// Core S7.2.1 - the application names its own conditions on this module; the
// library declares none. Safe-motion status (S9.2) is read-only application
// input, so "STO cleared" is declared here by the station that can see it.
// Declared conditions start FALSE: declaring one states an intent to gate.
METHOD DeclareCondition : BOOL
VAR_INPUT
    Index : INT;
    DescriptionKey : STRING(255);
    Reason : E_Reason;
    Bypassable : BOOL;
END_VAR
IF (Index < 1) OR (Index > PL_Fraktal.MAX_PERMINTLK_COND) THEN
    DeclareCondition := FALSE;
    RETURN;
END_IF
_appCond[Index] := FALSE;
DeclareCondition := Intlk.Define(Index := Index, Description := DescriptionKey,
    Reason := Reason, Bypassable := Bypassable);
END_METHOD

// Drive a condition declared by DeclareCondition, every scan.
METHOD SetCondition : BOOL
VAR_INPUT
    Index : INT;
    Ok : BOOL;
END_VAR
IF (Index < 1) OR (Index > PL_Fraktal.MAX_PERMINTLK_COND) THEN
    SetCondition := FALSE;
    RETURN;
END_IF
_appCond[Index] := Ok;
SetCondition := TRUE;
END_METHOD

// §7.6.1 held command - JOG_POS / JOG_NEG. Called EVERY SCAN while the
// operator holds the button; silence stops the axis (see _M_JogCyclic).
//
// This method only RECORDS the request. Nothing moves from here: the decision to
// drive is taken once per scan in _M_JogCyclic, where the interlock, the enabling
// device, the freshness deadline and the command handshake are all weighed
// together. Keeping the decision in one place is what makes it reviewable.
METHOD RequestHeldCommand : BOOL
VAR_INPUT
    Value  : DINT;
    Enable : ST_ManualEnableStatus;
END_VAR
// IF rather than CASE: a CASE label must be a compile-time constant, and
// TO_DINT(enum) is a call. The intent is the same - a defined ELSE (§5.6).
IF Value = TO_DINT(E_AxisCommand.JOG_POS) THEN
    _jogReqDir :=  1;
ELSIF Value = TO_DINT(E_AxisCommand.JOG_NEG) THEN
    _jogReqDir := -1;
ELSE
    // Not a held command of this type. Refuse, and do not record it - an unknown
    // value must never leave a stale direction behind.
    RequestHeldCommand := FALSE;
    RETURN;
END_IF

_jogSeen    := TRUE;
_jogEnabled := Enable.Held;

// Refused up front, with the reason, when no safety-rated enabling device is
// permitting. The axis ALSO has to pass its interlocks in _M_JogCyclic - this is
// an additional requirement, never a way around them (§9).
//
// StationCfg.JogRequiresEnable is what an installation WITHOUT an enabling
// device declares (§3.8a). It relaxes exactly this one requirement: the
// interlocks, the freshness deadline and the command handshake are untouched,
// so a station that declares it still cannot jog through a dropped interlock
// or on a stale request.
IF _station.JogRequiresEnable AND NOT Enable.Held THEN
    OutImm.JogStopReason := PL_ModuleReasons.AXIS_JOG_NOT_ENABLED;
    RequestHeldCommand := FALSE;
    RETURN;
END_IF
RequestHeldCommand := TRUE;
END_METHOD

// The one place a jog is allowed to start, continue, or stop. Runs every scan
// from OnCyclic, whether or not anybody asked - because "nobody asked" is
// precisely the condition that has to stop the axis.
METHOD PRIVATE _M_JogCyclic
VAR
    drive : BOOL;
END_VAR
// Freshness (O10). The timer accumulates while no request arrives, so a caller
// that goes quiet - operator released, HMI closed, network stalled with the
// button still down - stops the axis after JogTimeout. A few scans of jitter are
// tolerated; a dead transport is not.
_tJogStale(IN := NOT _jogSeen, PT := ParCfg.JogTimeout);

// Every gate that must hold for the axis to move by hand, in one expression so
// there is one place to review. Interlocks are NOT bypassed for teaching: the
// station is expected to have wired its guard condition so the safety system's
// teach grant satisfies it, and if it has not, the axis simply does not jog
// (§7.2.1, fail-closed).
drive := (_jogReqDir <> 0)
    AND NOT _tJogStale.Q
    AND (_jogEnabled OR NOT _station.JogRequiresEnable)
    AND Intlk.AllOk
    AND NOT Busy                        // a commanded move owns the axis (§6.1)
    AND __ISVALIDREF(_axis);

// Say why it stopped, once, on the transition. Published status, not an alarm.
IF _jogDriving AND NOT drive THEN
    // The PLC genuinely cannot tell "operator let go" from "link died" - both
    // are simply the request no longer arriving - so it reports what it knows
    // rather than inventing a distinction. The HMI CAN tell, because it knows
    // whether it is still sending, and surfaces the difference there.
    IF _tJogStale.Q THEN
        OutImm.JogStopReason := PL_ModuleReasons.AXIS_JOG_RELEASED;
    ELSIF NOT _jogEnabled AND _station.JogRequiresEnable THEN
        OutImm.JogStopReason := PL_ModuleReasons.AXIS_JOG_NOT_ENABLED;
    ELSIF NOT Intlk.AllOk THEN
        OutImm.JogStopReason := TO_DINT(E_Reason.INTERLOCK_DROPPED);
    ELSE
        OutImm.JogStopReason := PL_ModuleReasons.AXIS_JOG_RELEASED;
    END_IF
    _jogReqDir := 0;
END_IF

IF __ISVALIDREF(_axis) THEN
    _jogFb(Axis := _axis,
           JogForward   := drive AND (_jogReqDir > 0),
           JogBackwards  := drive AND (_jogReqDir < 0),
           Mode         := MC_JOGMODE_CONTINOUS,
           Velocity     := ParCfg.JogVelocity,
           Acceleration := ParCfg.JogAcceleration,
           Deceleration := ParCfg.Deceleration);
END_IF

_jogDriving    := drive;
OutImm.Jogging := drive;
_jogSeen       := FALSE;   // consumed: the caller must ask again next scan
END_METHOD

METHOD Setup : BOOL
VAR_INPUT
    Name    : STRING(80);
    AxisRef : REFERENCE TO AXIS_REF;
    Recipe  : I_RecipeProvider;
END_VAR
VAR
    InitialModel : ST_ModelId;
END_VAR
_M_SetName(Name);
_M_SetPresentation(DisplayNameKey := 'std.moduleType.axis.name', DescriptionKey := 'std.moduleType.axis.description', TypeKey := 'std.moduleType.axis');
_axis REF= AxisRef;                      // [TC3] TC3 S3.11
_recipe := Recipe;
// No Intlk.Define here: safe-motion status and station policy are the
// application's to name (S7.2.1).
_M_PublishCommand(Value := TO_DINT(E_AxisCommand.HOME), Label := 'std.command.home');
_M_PublishCommand(Value := TO_DINT(E_AxisCommand.MOVE_TO), Label := 'std.command.moveTo');
_M_PublishHeldCommand(Value := TO_DINT(E_AxisCommand.JOG_POS), Label := 'std.command.jogPositive');
_M_PublishHeldCommand(Value := TO_DINT(E_AxisCommand.JOG_NEG), Label := 'std.command.jogNegative');
Setup := PrepareRecipe(Model := InitialModel);
IF Setup THEN CommitRecipe(); END_IF

// §3.8b restore, in one call. The rule - version 0 is a first boot that lost
// nothing, any other unrecognized version means a real image was rejected and
// is annunciated with this module's own path - is written ONCE in
// FB_ModuleBase, because every module type with a StationCfg needs exactly it
// (§1.1 O1). This type supplies only the part that is genuinely its own: what
// its declared defaults are.
//
// The CONSEQUENCE of a loss is the deployment's, not this module's: the root
// applies E_ConfigRestorePolicy. Faulting the axis here, as this used to,
// forced BLOCK_UNTIL_ACKNOWLEDGED on every station that ever used an axis.
IF NOT M_RestoreStationCfg(pVersion := ADR(_station.SchemaVersion),
        SchemaVersion := AXIS_STATIONCFG_SCHEMA) THEN
    _station.TaughtPosition := 0.0;          // this type's declared default
    // The default is the SAFE reading: an axis that lost its configuration
    // requires an enabling device again, rather than inheriting a bench's
    // relaxation into a machine that never declared one.
    _station.JogRequiresEnable := TRUE;
END_IF

// §3.8a - the taught position is an ordinary editable value: typeable by an
// engineer who knows the number, and validated against the same soft limits
// whichever way it arrives.
Setup := M_RegisterConfigNumber(Key := 'axis.taughtPosition',
    Item := 'StationCfg/TaughtPosition', LabelKey := 'std.config.axisTaughtPosition',
    Unit := E_EngUnit.MILLIMETER, Kind := E_ConfigKind.STATION_CFG, Storage := E_ConfigStorage.AS_LREAL,
    pTarget := ADR(_station.TaughtPosition), Minimum := ParCfg.SoftMin, Maximum := ParCfg.SoftMax,
    RequiresReady := FALSE) AND Setup;

// §3.8c - and it can be DEMONSTRATED instead of typed: jog the axis to the
// position, then capture. The source is OutImm.ActPos, which this module already
// publishes, so the operator sees the number before storing it (§3.8c(b)).
Setup := M_RegisterCapture(WriteKey := 'axis.taughtPosition',
    pSource := ADR(OutImm.ActPos), SourceStorage := E_ConfigStorage.AS_LREAL) AND Setup;

// §3.8a - published as an editable capability so "does this installation have
// an enabling device?" is visible, audited and carried in a station parameter
// set, instead of being a silent assumption nobody can see.
Setup := M_RegisterConfigFlag(Key := 'axis.jogRequiresEnable',
    Item := 'StationCfg/JogRequiresEnable',
    LabelKey := 'std.config.axisJogRequiresEnable',
    Kind := E_ConfigKind.STATION_CFG, pTarget := ADR(_station.JogRequiresEnable),
    RequiresReady := TRUE) AND Setup;
END_METHOD

// §3.8a/§G.4a - declare whether this INSTALLATION has a safety-rated enabling
// device for manual motion. Called by the composition root; it also stamps the
// schema version forward, so a call made before Setup survives the restore
// (a matching version is restored as-is rather than defaulted).
//
// FALSE relaxes exactly one requirement - the enabling device - and nothing
// else: interlocks, the freshness deadline and the command handshake all still
// apply, and jog still refuses a stale request. A station that declares FALSE
// should declare a §7.5 engineering gate with it, so the machine says out loud
// that it is jogging without one.
METHOD SetJogRequiresEnable : BOOL
VAR_INPUT
    Required : BOOL;
END_VAR
_station.JogRequiresEnable := Required;
_station.SchemaVersion := AXIS_STATIONCFG_SCHEMA;
SetJogRequiresEnable := TRUE;
END_METHOD

// Functional stop used by an owning sequence on abort/interlock loss. This is a
// controlled MC_Stop, NOT a certified safe stop: the safety system remains
// authoritative and STO is its business, not this module's (S9).
METHOD WithdrawOutputs
IF __ISVALIDREF(_axis) THEN
    _moveFb(Axis := _axis, Execute := FALSE);
    _homeFb(Axis := _axis, Execute := FALSE);
    // A held jog is an output of this module like any other, so it is withdrawn
    // here too - otherwise an abort would stop the commanded move and leave a
    // jog running.
    _jogFb(Axis := _axis, JogForward := FALSE, JogBackwards := FALSE);
    _stopFb(Axis := _axis, Execute := TRUE, Deceleration := ParCfg.Deceleration);
END_IF
_jogReqDir  := 0;
_jogDriving := FALSE;
OutImm.Jogging := FALSE;
_tMove(IN := FALSE);
END_METHOD

METHOD PROTECTED OnAbort : DINT
OnAbort := SUPER^.OnAbort();            // base first (S3.14.2)
WithdrawOutputs();
END_METHOD

METHOD PrepareRecipe : BOOL
VAR_INPUT
    Model : ST_ModelId;
END_VAR
IF _recipe = 0 THEN
    _parCfgStaged := ParCfg;
    _recipePrepared := TRUE;
    PrepareRecipe := TRUE;
ELSIF _recipe.Load(ModelCode := Model.ModelCode, RecipeKey := 'AxisCM', pParCfg := ADR(_parCfgStaged), Size := SIZEOF(_parCfgStaged)) THEN
    _recipePrepared := TRUE;
    PrepareRecipe := TRUE;
ELSE
    _M_Fault(E_Reason.RECIPE_INVALID, 'std.error.recipeSchemaInvalid');
    _recipePrepared := FALSE;
    PrepareRecipe := FALSE;
END_IF
END_METHOD

METHOD CommitRecipe
IF _recipePrepared THEN ParCfg := _parCfgStaged; END_IF
_recipePrepared := FALSE;
END_METHOD

METHOD AbortRecipe
_recipePrepared := FALSE;
END_METHOD

// Stop the axis, THEN fault. _M_FaultN raises the reason without touching
// motion, so faulting mid-move would leave the drive commanded - the same defect
// the separator's _M_FaultClosed exists to prevent, and worse here because the
// load is moving.
METHOD PRIVATE _M_FaultStopped
VAR_INPUT
    Code : DINT;
    Text : STRING(255);
END_VAR
WithdrawOutputs();
_M_FaultN(Code := Code, Text := Text);
END_METHOD

METHOD PROTECTED _M_Dispatch
VAR
    dg : ST_Diagnostic;
END_VAR
IF _manualReq THEN
    _manualReq := FALSE;
    IF (_manualCmd = TO_DINT(E_AxisCommand.HOME)) OR (_manualCmd = TO_DINT(E_AxisCommand.MOVE_TO)) THEN
        Command := _manualCmd;
    ELSE
        _M_Fault(E_Reason.UNSUPPORTED_COMMAND, 'std.error.unsupportedAxisCommand');
        RETURN;
    END_IF
END_IF
IF (Command <> E_AxisCommand.HOME) AND (Command <> E_AxisCommand.MOVE_TO) THEN
    _M_Fault(E_Reason.UNSUPPORTED_COMMAND, 'std.error.unsupportedAxisCommand');
    RETURN;
END_IF
IF Command = E_AxisCommand.HOME THEN
    _M_TagCommand(Id := 1, Label := 'std.command.home');          // S8.11.4(a)
ELSE
    _M_TagCommand(Id := 2, Label := 'std.command.moveTo');
END_IF
_M_ApplyConditions();
Intlk();
IF NOT Intlk.AllOk THEN
    // HELD, not a fault (S6.1). Losing a declared condition mid-move is expected
    // - an operator releasing an enable is the designed way to stop. The axis is
    // brought to a controlled stop by the same permit that gates the enable, and
    // the move resumes from step 10 with a full MoveTimeout window so a hold
    // cannot silently consume travel time the axis was not moving for.
    WithdrawOutputs();
    dg := Intlk.Diagnostic;
    dg.SourcePath := _name;                          // owner sets the path (S7.2)
    _M_HoldDiag(Diag := dg);
    _step := 10;
    RETURN;
END_IF
IF Command = E_AxisCommand.HOME THEN
    _M_Home();
ELSE
    _M_MoveTo();
END_IF
END_METHOD

METHOD PRIVATE _M_Home
IF NOT __ISVALIDREF(_axis) THEN
    _M_FaultN(Code := PL_ModuleReasons.AXIS_DRIVE_FAULT, Text := 'std.error.axisNotBound');
    RETURN;
END_IF
CASE _step OF
    10:
        OutCmd.InPosition := FALSE;
        _homed := FALSE;                       // homing invalidates any previous datum
        _homeFb(Axis := _axis, Execute := FALSE);
        _tMove(IN := FALSE);
        _step := 20;
    20:
        _homeFb(Axis := _axis, Execute := TRUE, Position := 0.0, HomingMode := MC_DefaultHoming);
        _tMove(IN := TRUE, PT := ParCfg.HomeTimeout);
        IF _homeFb.Done THEN
            _homeFb(Axis := _axis, Execute := FALSE);
            _tMove(IN := FALSE);
            _homed := TRUE;
            _M_Complete();
        ELSIF _homeFb.Error THEN
            _M_FaultStopped(Code := PL_ModuleReasons.AXIS_DRIVE_FAULT, Text := 'std.error.axisDriveFault');
        ELSIF _homeFb.CommandAborted THEN
            // CommandAborted means another motion command took the axis, which is
            // an abort and not a defect - route it through the base's own abort
            // path rather than inventing a fault for it.
            AbortCommand();
        ELSIF _tMove.Q THEN
            _M_FaultStopped(Code := PL_ModuleReasons.AXIS_MOVE_TIMEOUT, Text := 'std.error.axisMoveTimeout');
        END_IF
ELSE
    _M_Fault(E_Reason.STEP_STALLED, 'std.error.undefinedStep');    // defined ELSE (S5.6)
END_CASE
END_METHOD

METHOD PRIVATE _M_MoveTo
// Validate the REQUEST before the STATE, and both before commanding motion
// (S5.6). Annex G checked homed-first; range-first is used here because a target
// outside the soft limits is malformed regardless of whether the axis is homed,
// and reporting "not homed" for an impossible target sends the operator to the
// wrong problem. It also makes both rejections provable without a licensed NC
// axis, since neither issues an MC_* call.
IF (ParCmd.Target < ParCfg.SoftMin) OR (ParCmd.Target > ParCfg.SoftMax) THEN
    _M_FaultN(Code := PL_ModuleReasons.AXIS_TARGET_OOR, Text := 'std.error.axisTargetOutOfRange');
    RETURN;
END_IF
IF NOT _homed THEN
    _M_FaultN(Code := PL_ModuleReasons.AXIS_NOT_HOMED, Text := 'std.error.axisNotHomed');
    RETURN;
END_IF
IF NOT __ISVALIDREF(_axis) THEN
    _M_FaultN(Code := PL_ModuleReasons.AXIS_DRIVE_FAULT, Text := 'std.error.axisNotBound');
    RETURN;
END_IF
CASE _step OF
    10:
        OutCmd.InPosition := FALSE;
        _moveFb(Axis := _axis, Execute := FALSE);
        _tMove(IN := FALSE);
        _step := 20;
    20:
        // MC_MoveAbsolute's Busy/Done/Error/CommandAborted map one-to-one onto
        // the CM handshake, which is what lets a parent Unit command MOVE_TO
        // exactly as it commands a cylinder EXTEND (S6.1).
        _moveFb(Axis := _axis, Execute := TRUE, Position := ParCmd.Target,
            Velocity := ParCfg.Velocity, Acceleration := ParCfg.Acceleration,
            Deceleration := ParCfg.Deceleration);
        _tMove(IN := TRUE, PT := ParCfg.MoveTimeout);
        IF _moveFb.Done THEN
            _moveFb(Axis := _axis, Execute := FALSE);
            _tMove(IN := FALSE);
            OutCmd.InPosition := TRUE;
            _M_Complete();
        ELSIF _moveFb.Error THEN
            _M_FaultStopped(Code := PL_ModuleReasons.AXIS_DRIVE_FAULT, Text := 'std.error.axisDriveFault');
        ELSIF _moveFb.CommandAborted THEN
            // CommandAborted means another motion command took the axis, which is
            // an abort and not a defect - route it through the base's own abort
            // path rather than inventing a fault for it.
            AbortCommand();
        ELSIF _tMove.Q THEN
            _M_FaultStopped(Code := PL_ModuleReasons.AXIS_MOVE_TIMEOUT, Text := 'std.error.axisMoveTimeout');
        END_IF
ELSE
    _M_Fault(E_Reason.STEP_STALLED, 'std.error.undefinedStep');
END_CASE
END_METHOD

END_FUNCTION_BLOCK

// ---- FB_SeparatorCM.TcPOU
// Annex A worked example on the base class: the type is ONLY its device logic.
//
// It defines NO interlocks of its own, deliberately. Core S7.2.1 confines a
// reusable library to "device-intrinsic conditions or explicitly injected generic
// policy", and none of Annex A's four published conditions qualify: area-safe is
// a S9.2 safety alias, air pressure is a utility, jam is a flag that is not even
// on this device's HAL, and downstream-ready is line policy. All four belong to
// the owning Unit's Release/Permissives object (S7.2.1, S4.2).
//
// So the application declares and drives them through DeclareCondition/
// SetCondition. They land in this module's own FB_PermIntlk, which keeps the
// provenance S7.2.1 requires - first-out, release report and HMI drill-down all
// read the same ST_IntlkCond records - without the library naming policy it
// cannot see. A per-condition setter was rejected: FB_CylinderCM.SetAreaSafe is
// exactly that shape and no application has ever called it.
FUNCTION_BLOCK FB_SeparatorCM EXTENDS FB_ControlModuleBase
VAR_INPUT
    Command : E_SeparatorCommand;
    ParCfg : ST_SeparatorParCfg;
    ParCmd : ST_SeparatorParCmd;
END_VAR
VAR_OUTPUT
    OutCmd : ST_SeparatorOutCmd;
    OutImm : ST_SeparatorOutImm;
    Intlk  : FB_PermIntlk;
END_VAR
VAR
    {attribute 'OPC.UA.DA' := '0'}
    _hal    : REFERENCE TO ST_SeparatorHal;
    {attribute 'OPC.UA.DA' := '0'}
    _recipe : I_RecipeProvider;
    _tPhase : TON;                       // per-phase timeout (open / clear / arrive)
    _tClose : TON;                       // close delay
    _parCfgStaged : ST_SeparatorParCfg;
    _recipePrepared : BOOL;
    // Application-owned conditions (S7.2.1). Declared FALSE so a declared-but-
    // undriven condition holds the module rather than silently permitting it.
    _appCond : ARRAY[1..PL_Fraktal.MAX_PERMINTLK_COND] OF BOOL;
END_VAR

Cyclic();

METHOD PROTECTED OnCyclic : DINT
OnCyclic := SUPER^.OnCyclic();
// Re-drive every application condition each scan, so a manual command obeys the
// same rule as a sequenced one (S7.2).
_M_ApplyConditions();
Intlk();
IF __ISVALIDREF(_hal) THEN              // defensive (S5.6) [TC3]
    OutImm.CarrierAt    := _hal.CarrierAt;
    OutImm.CarrierAfter := _hal.CarrierAfter;
    OutImm.OpenedFb     := _hal.OpenedFb;
    OutImm.ValveOpen    := _hal.ValveOpen;
    OutCmd.SeparatorOpen := _hal.ValveOpen;
END_IF
END_METHOD

METHOD PRIVATE _M_ApplyConditions
VAR
    i : INT;
END_VAR
FOR i := 1 TO PL_Fraktal.MAX_PERMINTLK_COND DO
    Intlk.Cond[i] := _appCond[i];
END_FOR
END_METHOD

// Core S7.2.1 - the application names its own conditions on this module.
// The library defines none, so every index is the application's to claim.
// Returns FALSE on an out-of-range index rather than silently ignoring it (S5.6).
//
// Declared conditions start FALSE: declaring one states an intent to gate, so
// the fail-closed default is to hold until the application drives it. A station
// that wants no gate simply declares nothing.
METHOD DeclareCondition : BOOL
VAR_INPUT
    Index : INT;
    DescriptionKey : STRING(255);
    Reason : E_Reason;
    Bypassable : BOOL;
END_VAR
IF (Index < 1) OR (Index > PL_Fraktal.MAX_PERMINTLK_COND) THEN
    DeclareCondition := FALSE;
    RETURN;
END_IF
_appCond[Index] := FALSE;
DeclareCondition := Intlk.Define(Index := Index, Description := DescriptionKey,
    Reason := Reason, Bypassable := Bypassable);
END_METHOD

// Drive a condition declared by DeclareCondition. Call it every scan from the
// owning Unit's Release object; the value is re-applied in OnCyclic so dispatch
// and the release report always read the same state.
METHOD SetCondition : BOOL
VAR_INPUT
    Index : INT;
    Ok : BOOL;
END_VAR
IF (Index < 1) OR (Index > PL_Fraktal.MAX_PERMINTLK_COND) THEN
    SetCondition := FALSE;
    RETURN;
END_IF
_appCond[Index] := Ok;
SetCondition := TRUE;
END_METHOD

METHOD Setup : BOOL
VAR_INPUT
    Name   : STRING(80);
    HalRef : REFERENCE TO ST_SeparatorHal;
    Recipe : I_RecipeProvider;
END_VAR
VAR
    InitialModel : ST_ModelId;
END_VAR
_M_SetName(Name);
_M_SetPresentation(DisplayNameKey := 'std.moduleType.separator.name', DescriptionKey := 'std.moduleType.separator.description', TypeKey := 'std.moduleType.separator');
_hal REF= HalRef;                        // [TC3] TC3 S3.11
_recipe := Recipe;
// No Intlk.Define here: this type publishes no condition it cannot itself
// derive (S7.2.1). The application declares its own via DeclareCondition.
_M_PublishCommand(Value := TO_DINT(E_SeparatorCommand.SEPARATE), Label := 'std.command.separate');
_M_PublishCommand(Value := TO_DINT(E_SeparatorCommand.OPEN_CLOSE), Label := 'std.command.openClose');
Setup := PrepareRecipe(Model := InitialModel);
IF Setup THEN CommitRecipe(); END_IF
END_METHOD

// Functional stop used by an owning sequence on abort/interlock loss.
// This is not a certified stop; the safety system remains authoritative (S9).
METHOD WithdrawOutputs
IF __ISVALIDREF(_hal) THEN
    _hal.ValveOpen := FALSE;
END_IF
END_METHOD

METHOD PROTECTED OnAbort : DINT
OnAbort := SUPER^.OnAbort();            // base first (S3.14.2)
IF __ISVALIDREF(_hal) THEN
    _hal.ValveOpen := FALSE;
END_IF
END_METHOD

METHOD PrepareRecipe : BOOL
VAR_INPUT
    Model : ST_ModelId;
END_VAR
IF _recipe = 0 THEN
    _parCfgStaged := ParCfg;
    _recipePrepared := TRUE;
    PrepareRecipe := TRUE;
ELSIF _recipe.Load(ModelCode := Model.ModelCode, RecipeKey := 'SeparatorCM', pParCfg := ADR(_parCfgStaged), Size := SIZEOF(_parCfgStaged)) THEN
    _recipePrepared := TRUE;
    PrepareRecipe := TRUE;
ELSE
    _M_Fault(E_Reason.RECIPE_INVALID, 'std.error.recipeSchemaInvalid');
    _recipePrepared := FALSE;
    PrepareRecipe := FALSE;
END_IF
END_METHOD

METHOD CommitRecipe
IF _recipePrepared THEN ParCfg := _parCfgStaged; END_IF
_recipePrepared := FALSE;
END_METHOD

METHOD AbortRecipe
_recipePrepared := FALSE;
END_METHOD

METHOD PROTECTED _M_Dispatch
VAR
    dg : ST_Diagnostic;
END_VAR
IF _manualReq THEN
    _manualReq := FALSE;
    IF (_manualCmd = TO_DINT(E_SeparatorCommand.SEPARATE)) OR (_manualCmd = TO_DINT(E_SeparatorCommand.OPEN_CLOSE)) THEN
        Command := _manualCmd;
    ELSE
        _M_Fault(E_Reason.UNSUPPORTED_COMMAND, 'std.error.unsupportedSeparatorCommand');
        RETURN;
    END_IF
END_IF
IF (Command <> E_SeparatorCommand.SEPARATE) AND (Command <> E_SeparatorCommand.OPEN_CLOSE) THEN
    _M_Fault(E_Reason.UNSUPPORTED_COMMAND, 'std.error.unsupportedSeparatorCommand');
    RETURN;
END_IF
IF Command = E_SeparatorCommand.SEPARATE THEN
    _M_TagCommand(Id := 1, Label := 'std.command.separate');      // S8.11.4(a)
ELSE
    _M_TagCommand(Id := 2, Label := 'std.command.openClose');
END_IF
_M_ApplyConditions();
Intlk();
IF NOT Intlk.AllOk THEN
    // HELD, not a fault (S6.1): an interlock is a condition that must hold DURING
    // the action, and losing one is often expected - the same reasoning as
    // FB_CylinderCM. Outputs are withdrawn here by the same permit that gates
    // them; only the classification and the way out differ. Rewinding to step 10
    // re-arms the phase timer with a full window, so a hold cannot silently
    // consume travel time the carrier was not moving for.
    IF __ISVALIDREF(_hal) THEN
        _hal.ValveOpen := FALSE;
    END_IF
    _tPhase(IN := FALSE);
    dg := Intlk.Diagnostic;
    dg.SourcePath := _name;                          // owner sets the path (S7.2)
    _M_HoldDiag(Diag := dg);
    _step := 10;
    RETURN;
END_IF
IF Command = E_SeparatorCommand.OPEN_CLOSE THEN
    _M_OpenClose();
    RETURN;
END_IF
// ---- SEPARATE: release exactly one carrier (Annex A) ----------------------
CASE _step OF
    10:                                  // open, and require a carrier present
        OutCmd.SeparateOk := FALSE;
        _hal.ValveOpen := TRUE;
        _tPhase(IN := TRUE, PT := ParCfg.MaxOpenTime);
        IF _hal.CarrierAt THEN
            _tPhase(IN := FALSE);
            _step := 20;
        ELSIF _tPhase.Q THEN
            _tPhase(IN := FALSE);
            _M_FaultClosed(Code := PL_ModuleReasons.SEP_NO_CARRIER_AT, Text := 'std.error.separatorNoCarrierAt');
        END_IF
    20:                                  // the carrier must clear CarrierAt
        _tPhase(IN := TRUE, PT := ParCfg.MaxOpenTime);
        IF NOT _hal.CarrierAt THEN
            _tPhase(IN := FALSE);
            IF ParCfg.CheckAfter THEN _step := 30; ELSE _step := 40; END_IF
        ELSIF _tPhase.Q THEN
            _tPhase(IN := FALSE);
            _M_FaultClosed(Code := PL_ModuleReasons.SEP_CARRIER_NOT_CLEARED, Text := 'std.error.separatorCarrierNotCleared');
        END_IF
    30:                                  // arrival check past the separator
        _tPhase(IN := TRUE, PT := ParCfg.SOnMaxTime);
        IF _hal.CarrierAfter THEN
            _tPhase(IN := FALSE);
            _step := 40;
        ELSIF _tPhase.Q THEN
            _tPhase(IN := FALSE);
            _M_FaultClosed(Code := PL_ModuleReasons.SEP_CARRIER_NOT_ARRIVED, Text := 'std.error.separatorCarrierNotArrived');
        END_IF
    40:                                  // close after the configured delay
        _tClose(IN := TRUE, PT := ParCfg.CloseDelay);
        IF _tClose.Q OR (ParCfg.CloseDelay = T#0S) THEN
            _tClose(IN := FALSE);
            _hal.ValveOpen := FALSE;
            IF ParCfg.CheckAfter THEN
                _tPhase(IN := TRUE, PT := ParCfg.SOnMaxTime);
                _step := 50;
            ELSE
                OutCmd.SeparateOk := TRUE;
                _M_Complete();
            END_IF
        END_IF
    50:                                  // the carrier must clear CarrierAfter
        _tPhase(IN := TRUE, PT := ParCfg.SOnMaxTime);
        IF NOT _hal.CarrierAfter THEN
            _tPhase(IN := FALSE);
            OutCmd.SeparateOk := TRUE;
            _M_Complete();
        ELSIF _tPhase.Q THEN
            _tPhase(IN := FALSE);
            _M_FaultClosed(Code := PL_ModuleReasons.SEP_SON_NOT_CLEARED, Text := 'std.error.separatorSonNotCleared');
        END_IF
ELSE
    _M_Fault(E_Reason.STEP_STALLED, 'std.error.undefinedStep');    // defined ELSE (S5.6)
END_CASE
END_METHOD

METHOD PRIVATE _M_OpenClose
// Hold the stopper open or closed. Closing is immediate; opening optionally
// confirms the feedback when the station has wired one (ParCfg.UsesOpenFb).
_hal.ValveOpen := ParCmd.OpenStopper;
IF NOT ParCmd.OpenStopper THEN
    _tPhase(IN := FALSE);
    _M_Complete();
    RETURN;
END_IF
IF NOT ParCfg.UsesOpenFb THEN
    _tPhase(IN := FALSE);
    _M_Complete();
    RETURN;
END_IF
_tPhase(IN := TRUE, PT := ParCfg.MaxOpenTime);
IF _hal.OpenedFb THEN
    _tPhase(IN := FALSE);
    _M_Complete();
ELSIF _tPhase.Q THEN
    _tPhase(IN := FALSE);
    _M_FaultClosed(Code := PL_ModuleReasons.SEP_NOT_OPENED_FB, Text := 'std.error.separatorNotOpenedFb');
END_IF
END_METHOD

// Withdraw the valve, THEN fault. _M_FaultN only raises the reason; it does not
// touch outputs, so faulting from an open phase would leave the stopper
// energised while the module reported ERROR. Annex A faults and closes in one
// step for exactly this reason, and a separator that stays open on a fault
// keeps releasing carriers it can no longer account for.
METHOD PRIVATE _M_FaultClosed
VAR_INPUT
    Code : DINT;
    Text : STRING(255);
END_VAR
WithdrawOutputs();
_M_FaultN(Code := Code, Text := Text);
END_METHOD

END_FUNCTION_BLOCK

// ---- FB_ConfigurableCylinderCM.TcPOU
// Production-grade basic pneumatic cylinder Control Module (Core §2.2 base) with
// OPTIONAL and REDUNDANT position sensors (safety cylinders). Per position: 0..N
// sensors; 0 = sensorless (time-based). 'Arrived' = ALL present sensors TRUE (AND,
// safest); a persistent split of redundant sensors faults (discrepancy monitoring).
// The type is ONLY its device logic; lifecycle/timing/first-out/abort are inherited.
FUNCTION_BLOCK FB_ConfigurableCylinderCM EXTENDS FB_ControlModuleBase
VAR_INPUT
    Command : E_ConfigurableCylinderCommand;
    ParCfg : ST_ConfigurableCylinderParCfg;
    ParCmd : ST_ConfigurableCylinderParCmd;
END_VAR
VAR_OUTPUT
    OutCmd : ST_ConfigurableCylinderOutCmd;
    OutImm : ST_ConfigurableCylinderOutImm;
    Intlk  : FB_PermIntlk;
END_VAR
VAR
    {attribute 'OPC.UA.DA' := '0'}
    _hal     : REFERENCE TO ST_ConfigurableCylinderHal;
    {attribute 'OPC.UA.DA' := '0'}
    _recipe  : I_RecipeProvider;
    _tMove   : TON;
    _tSettle : TON;
    _tDiscH  : TON;                             // home discrepancy timer
    _tDiscW  : TON;                             // work discrepancy timer
    _cfgOk   : BOOL;
    _areaSafe : BOOL := TRUE;                   // §7.2 application-supplied area/process interlock
    _areaSafeKey : STRING(255);
    _parCfgStaged : ST_ConfigurableCylinderParCfg;
    _recipePrepared : BOOL;
END_VAR

Cyclic();

METHOD Setup : BOOL
VAR_INPUT
    Name   : STRING(80);
    HalRef : REFERENCE TO ST_ConfigurableCylinderHal;
    Recipe : I_RecipeProvider;
END_VAR
VAR
    InitialModel : ST_ModelId;
END_VAR
_M_SetName(Name);
_M_SetPresentation(DisplayNameKey := 'std.moduleType.configurableCylinder.name', DescriptionKey := 'std.moduleType.configurableCylinder.description', TypeKey := 'std.moduleType.configurableCylinder');
_M_PublishCommand(Value := TO_DINT(E_ConfigurableCylinderCommand.TO_HOME), Label := 'std.command.toHome');   // §7.6.1 catalog
_M_PublishCommand(Value := TO_DINT(E_ConfigurableCylinderCommand.TO_WORK), Label := 'std.command.toWork');
_hal REF= HalRef;                                        // [TC3] TC3 §3.11
_recipe := Recipe;
Intlk.Define(Index := 1, Description := 'std.interlock.areaSafe', Reason := E_Reason.INTERLOCK_DROPPED, Bypassable := FALSE);
Setup := PrepareRecipe(Model := InitialModel);
IF Setup THEN CommitRecipe(); END_IF
END_METHOD

METHOD PrepareRecipe : BOOL
VAR_INPUT
    Model : ST_ModelId;
END_VAR
_parCfgStaged := ParCfg;
IF _recipe <> 0 THEN
    IF NOT _recipe.Load(ModelCode := Model.ModelCode, RecipeKey := 'ConfigurableCylinderCM', pParCfg := ADR(_parCfgStaged), Size := SIZEOF(_parCfgStaged)) THEN
        _M_Fault(E_Reason.RECIPE_INVALID, 'std.error.recipeSchemaInvalid');
        PrepareRecipe := FALSE;
        RETURN;
    END_IF
END_IF
// counts within [0..MAX]; sensorless direction needs a usable travel time
_cfgOk := (_parCfgStaged.HomeSensorCount >= 0) AND (_parCfgStaged.HomeSensorCount <= PL_Fraktal.MAX_POS_SENSORS)
      AND (_parCfgStaged.WorkSensorCount >= 0) AND (_parCfgStaged.WorkSensorCount <= PL_Fraktal.MAX_POS_SENSORS)
      AND (_parCfgStaged.TravelTime < _parCfgStaged.MoveTimeout)
      AND ((_parCfgStaged.HomeSensorCount > 0) OR (_parCfgStaged.TravelTime > T#0S))
      AND ((_parCfgStaged.WorkSensorCount > 0) OR (_parCfgStaged.TravelTime > T#0S));
IF NOT _cfgOk THEN
    _M_FaultN(PL_ModuleReasons.CYL_CFG_INVALID, 'std.error.cylinderConfigurationInvalid');
    PrepareRecipe := FALSE;
    RETURN;
END_IF
_recipePrepared := TRUE;
PrepareRecipe := TRUE;
END_METHOD

METHOD CommitRecipe
IF _recipePrepared THEN ParCfg := _parCfgStaged; END_IF
_recipePrepared := FALSE;
END_METHOD

METHOD AbortRecipe
_recipePrepared := FALSE;
END_METHOD

// TRUE iff EVERY wired sensor for the position reads TRUE (AND-combine, safest).
// Count = 0 -> not sensor-decided (caller uses the time path).
METHOD PROTECTED _M_PosArrived : BOOL
VAR_INPUT
    Work : BOOL;    // TRUE = work position, FALSE = home
END_VAR
VAR
    i, n : INT;
    all  : BOOL;
END_VAR
n := SEL(Work, ParCfg.HomeSensorCount, ParCfg.WorkSensorCount);
IF n <= 0 THEN
    _M_PosArrived := FALSE;      // no sensors: caller must use the time-based path
    RETURN;
END_IF
all := TRUE;
FOR i := 1 TO n DO
    IF Work THEN
        IF NOT _hal.WorkFb[i] THEN all := FALSE; END_IF
    ELSE
        IF NOT _hal.HomeFb[i] THEN all := FALSE; END_IF
    END_IF
END_FOR
_M_PosArrived := all;
END_METHOD

// TRUE iff the position's redundant sensors DISAGREE (at least one TRUE and at
// least one FALSE) — the discrepancy condition. Single/zero sensor => never split.
METHOD PROTECTED _M_PosSplit : BOOL
VAR_INPUT
    Work : BOOL;
END_VAR
VAR
    i, n : INT;
    anyT, anyF : BOOL;
END_VAR
n := SEL(Work, ParCfg.HomeSensorCount, ParCfg.WorkSensorCount);
IF n < 2 THEN
    _M_PosSplit := FALSE;
    RETURN;
END_IF
FOR i := 1 TO n DO
    IF Work THEN
        IF _hal.WorkFb[i] THEN anyT := TRUE; ELSE anyF := TRUE; END_IF
    ELSE
        IF _hal.HomeFb[i] THEN anyT := TRUE; ELSE anyF := TRUE; END_IF
    END_IF
END_FOR
_M_PosSplit := anyT AND anyF;
END_METHOD

// live position resolve + discrepancy monitoring (both positions, every scan)
METHOD PROTECTED OnCyclic : DINT
OnCyclic := SUPER^.OnCyclic();
Intlk.Cond[1] := _areaSafe;
Intlk();
IF NOT __ISVALIDREF(_hal) THEN
    RETURN;
END_IF
OutImm.AtHome := (ParCfg.HomeSensorCount > 0) AND _M_PosArrived(Work := FALSE);
OutImm.AtWork := (ParCfg.WorkSensorCount > 0) AND _M_PosArrived(Work := TRUE);

// discrepancy monitoring — a persistent split of redundant sensors is a fault
_tDiscH(IN := _M_PosSplit(Work := FALSE), PT := ParCfg.DiscrepancyTime);
_tDiscW(IN := _M_PosSplit(Work := TRUE),  PT := ParCfg.DiscrepancyTime);
IF (_tDiscH.Q OR _tDiscW.Q) AND (_exec <> E_ExecState.ERROR) THEN
    _M_FaultN(PL_ModuleReasons.CYL_DISCREPANCY, 'std.error.cylinderSensorDiscrepancy');
END_IF

// resolve position (AtHome/AtWork already AND-combined)
IF OutImm.AtHome AND OutImm.AtWork THEN
    OutImm.Position := E_CylinderPosition.UNKNOWN;
ELSIF OutImm.AtHome THEN OutImm.Position := E_CylinderPosition.HOME;
ELSIF OutImm.AtWork THEN OutImm.Position := E_CylinderPosition.WORK;
ELSIF (ParCfg.HomeSensorCount > 0) OR (ParCfg.WorkSensorCount > 0) THEN OutImm.Position := E_CylinderPosition.MID;
END_IF

// both-positions-active plausibility while idle
IF (_exec = E_ExecState.READY) AND OutImm.AtHome AND OutImm.AtWork THEN
    _M_FaultN(PL_ModuleReasons.CYL_POS_IMPLAUSIBLE, 'std.error.cylinderPositionImplausible');
END_IF
END_METHOD

// §3.14.2 — fail-safe abort
METHOD PROTECTED OnAbort : DINT
OnAbort := SUPER^.OnAbort();
IF NOT __ISVALIDREF(_hal) THEN
    RETURN;
END_IF
IF ParCfg.DeenergizeOnAbort THEN
    _hal.ToWorkOut := FALSE;
    _hal.ToHomeOut := FALSE;
ELSIF ParCfg.SafePosOnAbort = E_CylinderPosition.WORK THEN
    _hal.ToWorkOut := TRUE;  _hal.ToHomeOut := FALSE;
ELSE
    _hal.ToWorkOut := FALSE; _hal.ToHomeOut := NOT ParCfg.SingleActing;
END_IF
END_METHOD

// Core §7.2/§7.2.1 — the application supplies this type's area/process interlock,
// the same shape as SetDirectionalPermits: a method (not an OPC UA write), and the
// condition is re-evaluated every scan so a manual command obeys the same rule.
//
// This replaces a SIM-only force hook that used to drive Cond[1] directly. That
// hook was the ONLY writer of the condition, so the slot an operator sees as
// "area safe" could be moved by a test and by nothing else: a reusable type
// published an interlock its application had no way to supply (§7.2.1), and the
// bypass shipped in every release build (§5.7). Driving the real condition is
// also strictly better test evidence - T3 now exercises the shipped path.
//
// Defaults TRUE: a station that declares no area interlock is not gated by one.
METHOD SetAreaSafe
VAR_INPUT
    Ok : BOOL;
    DescriptionKey : STRING(255);
END_VAR
_areaSafe := Ok;
_areaSafeKey := DescriptionKey;
IF _areaSafeKey <> '' THEN
    Intlk.Define(Index := 1, Description := _areaSafeKey, Reason := E_Reason.INTERLOCK_DROPPED, Bypassable := FALSE);
ELSE
    ;
END_IF
END_METHOD

// drive -> await (all-sensors-agree, or time when sensorless) -> settle -> done
METHOD PROTECTED _M_Dispatch
VAR
    toWork  : BOOL;
    n       : INT;
    arrived : BOOL;
    d       : ST_Diagnostic;
END_VAR
IF _manualReq THEN
    _manualReq := FALSE;                        // §7.6.1: apply the manual command value
    Command := _manualCmd;                      // routed THROUGH dispatch — interlocks still apply
END_IF
IF (Command <> E_ConfigurableCylinderCommand.TO_HOME) AND (Command <> E_ConfigurableCylinderCommand.TO_WORK) THEN
    _M_Fault(E_Reason.UNSUPPORTED_COMMAND, 'std.error.unsupportedCylinderCommand');
    RETURN;
END_IF
IF Command = E_ConfigurableCylinderCommand.TO_WORK THEN
    _M_TagCommand(Id := 2, Label := 'std.command.toWork');
    toWork := TRUE;
ELSE
    _M_TagCommand(Id := 1, Label := 'std.command.toHome');
    toWork := FALSE;
END_IF
IF NOT Intlk.AllOk THEN
    _hal.ToWorkOut := FALSE;
    _hal.ToHomeOut := FALSE;
    d := Intlk.Diagnostic;
    d.SourcePath := _name;
    _M_FaultDiag(d);
    RETURN;
END_IF
n := SEL(toWork, ParCfg.HomeSensorCount, ParCfg.WorkSensorCount);   // sensors on the TARGET position
CASE _step OF
    10:
        OutCmd.ReachedPosition := E_CylinderPosition.UNKNOWN;
        _hal.ToWorkOut := toWork;
        _hal.ToHomeOut := (NOT toWork) AND (NOT ParCfg.SingleActing);
        _tMove(IN := FALSE);
        _tSettle(IN := FALSE);
        _step := 20;
    20:  // await arrival
        _tMove(IN := TRUE, PT := ParCfg.MoveTimeout);
        IF n > 0 THEN
            arrived := _M_PosArrived(Work := toWork);        // ALL sensors agree
        ELSE
            _tSettle(IN := TRUE, PT := ParCfg.TravelTime);      // sensorless -> travel time
            arrived := _tSettle.Q;
        END_IF
        IF arrived THEN
            _tSettle(IN := FALSE);
            _step := 30;
        ELSIF _tMove.Q THEN
            _tMove(IN := FALSE);
            _M_FaultN(SEL(toWork, PL_ModuleReasons.CYL_HOME_NOT_REACHED, PL_ModuleReasons.CYL_WORK_NOT_REACHED),
                      SEL(toWork, 'std.error.cylinderHomeTimeout', 'std.error.cylinderWorkTimeout'));
        END_IF
    30:  // settle/debounce; re-confirm all sensors still agree
        _tSettle(IN := TRUE, PT := ParCfg.SettleTime);
        IF n <= 0 THEN
            OutCmd.ReachedPosition := SEL(toWork, E_CylinderPosition.HOME, E_CylinderPosition.WORK);
            _M_Complete();
        ELSIF _M_PosArrived(Work := toWork) THEN
            IF _tSettle.Q THEN
                OutCmd.ReachedPosition := SEL(toWork, E_CylinderPosition.HOME, E_CylinderPosition.WORK);
                _M_Complete();
            END_IF
        ELSE
            _tSettle(IN := FALSE);
            _step := 20;                                     // lost agreement; keep waiting in MoveTimeout
        END_IF
ELSE
    _M_Fault(E_Reason.STEP_STALLED, 'std.error.undefinedStep');
END_CASE
END_METHOD

PROPERTY AtPos : E_CylinderPosition
GET
AtPos := OutImm.Position;
END_GET
END_PROPERTY

END_FUNCTION_BLOCK

// ---- FB_ConfigurableCylinderSim.TcPOU
// §5.7 sim plant for FB_ConfigurableCylinderCM with redundant sensors: after a travel time
// it sets all HomeFb[1..HomeN] / WorkFb[1..WorkN] together. StuckWork[i]/StuckHome[i]
// pin a sensor OFF so a test can inject a discrepancy.
FUNCTION_BLOCK FB_ConfigurableCylinderSim
VAR_INPUT
    Travel : TIME := T#100MS;
    HomeN  : INT := 1;
    WorkN  : INT := 1;
    StuckHome : ARRAY[1..PL_Fraktal.MAX_POS_SENSORS] OF BOOL;   // TRUE = pin this sensor OFF
    StuckWork : ARRAY[1..PL_Fraktal.MAX_POS_SENSORS] OF BOOL;
END_VAR
VAR
    {attribute 'OPC.UA.DA' := '0'}
    _hal : REFERENCE TO ST_ConfigurableCylinderHal;
    _tW, _tH : TON;
    i : INT;
END_VAR

IF NOT __ISVALIDREF(_hal) THEN
    RETURN;
END_IF
_tW(IN := _hal.ToWorkOut, PT := Travel);
IF _tW.Q THEN
    FOR i := 1 TO WorkN DO _hal.WorkFb[i] := NOT StuckWork[i]; END_FOR
    FOR i := 1 TO HomeN DO _hal.HomeFb[i] := FALSE; END_FOR
END_IF
_tH(IN := _hal.ToHomeOut OR (NOT _hal.ToWorkOut AND NOT _hal.ToHomeOut), PT := Travel);
IF _tH.Q THEN
    FOR i := 1 TO HomeN DO _hal.HomeFb[i] := NOT StuckHome[i]; END_FOR
    FOR i := 1 TO WorkN DO _hal.WorkFb[i] := FALSE; END_FOR
END_IF

METHOD Setup : BOOL
VAR_INPUT
    HalRef : REFERENCE TO ST_ConfigurableCylinderHal;
    TravelTime : TIME;
    Home : INT;
    Work : INT;
END_VAR
VAR
    j : INT;
END_VAR
_hal REF= HalRef;
Travel := TravelTime;
HomeN := Home;
WorkN := Work;
FOR j := 1 TO HomeN DO _hal.HomeFb[j] := TRUE; END_FOR   // start at home, all agree
Setup := TRUE;
END_METHOD

END_FUNCTION_BLOCK

// ---- FB_ClampEM.TcPOU
// Annex B on the EM base: orchestration only, no device logic (§3.5); rollup §8.2.
FUNCTION_BLOCK FB_ClampEM EXTENDS FB_EquipmentModuleBase
VAR_INPUT
    Command : E_ClampCommand;
    ParCfg : ST_ClampParCfg;
    ParCmd : ST_ClampParCmd;
END_VAR
VAR_OUTPUT
    CylA, CylB : FB_CylinderCM;
    OutCmd : ST_ClampOutCmd;
    OutImm : ST_ClampOutImm;
END_VAR
VAR
    {attribute 'OPC.UA.DA' := '0'}
    _recipe : I_RecipeProvider;
    _tSettle : TON;
    _parCfgStaged : ST_ClampParCfg;
    _recipePrepared : BOOL;
END_VAR

Cyclic();

METHOD PROTECTED OnCyclic : DINT
OnCyclic := SUPER^.OnCyclic();
_M_TickChildren();                       // children stay live (Annex B §B.3)
END_METHOD

METHOD PrepareRecipe : BOOL
VAR_INPUT
    Model : ST_ModelId;
END_VAR
IF _recipe = 0 THEN
    _parCfgStaged := ParCfg;
    _recipePrepared := TRUE;
ELSIF _recipe.Load(ModelCode := Model.ModelCode, RecipeKey := 'ClampEM', pParCfg := ADR(_parCfgStaged), Size := SIZEOF(_parCfgStaged)) THEN
    _recipePrepared := TRUE;
ELSE
    _M_Fault(E_Reason.RECIPE_INVALID, 'std.error.recipeSchemaInvalid');
    _recipePrepared := FALSE;
    PrepareRecipe := FALSE;
    RETURN;
END_IF
PrepareRecipe := SUPER^.PrepareRecipe(Model := Model);
IF NOT PrepareRecipe THEN _recipePrepared := FALSE; END_IF
END_METHOD

METHOD CommitRecipe
SUPER^.CommitRecipe();
IF _recipePrepared THEN ParCfg := _parCfgStaged; END_IF
_recipePrepared := FALSE;
END_METHOD

METHOD AbortRecipe
SUPER^.AbortRecipe();
_recipePrepared := FALSE;
END_METHOD

METHOD Setup : BOOL
VAR_INPUT
    Name : STRING(80);
    HalA : REFERENCE TO ST_CylinderHal;
    HalB : REFERENCE TO ST_CylinderHal;
    Recipe : I_RecipeProvider;
END_VAR
VAR
    InitialModel : ST_ModelId;
END_VAR
_M_SetName(Name);
_M_SetPresentation(DisplayNameKey := 'std.moduleType.clamp.name', DescriptionKey := 'std.moduleType.clamp.description', TypeKey := 'std.moduleType.clamp');
_recipe := Recipe;
CylA.Setup(Name := CONCAT(Name, '.CylA'), HalRef := HalA, Recipe := Recipe);
CylB.Setup(Name := CONCAT(Name, '.CylB'), HalRef := HalB, Recipe := Recipe);
_M_Register(CylA);
_M_Register(CylB);
_M_PublishCommand(Value := TO_DINT(E_ClampCommand.CLAMP), Label := 'std.command.clamp');
_M_PublishCommand(Value := TO_DINT(E_ClampCommand.UNCLAMP), Label := 'std.command.unclamp');
Setup := PrepareRecipe(Model := InitialModel);
IF Setup THEN CommitRecipe(); END_IF
END_METHOD

METHOD PROTECTED _M_Dispatch
VAR
    dir : E_CylinderCommand;
    ext : BOOL;
END_VAR
IF _manualReq THEN
    _manualReq := FALSE;
    IF (_manualCmd = TO_DINT(E_ClampCommand.CLAMP)) OR (_manualCmd = TO_DINT(E_ClampCommand.UNCLAMP)) THEN
        Command := _manualCmd;
    ELSE
        _M_Fault(E_Reason.UNSUPPORTED_COMMAND, 'std.error.unsupportedClampCommand');
        RETURN;
    END_IF
END_IF
IF (Command <> E_ClampCommand.CLAMP) AND (Command <> E_ClampCommand.UNCLAMP) THEN
    _M_Fault(E_Reason.UNSUPPORTED_COMMAND, 'std.error.unsupportedClampCommand');
    RETURN;
END_IF
ext := (Command = E_ClampCommand.CLAMP);
dir := SEL(ext, E_CylinderCommand.RETRACT, E_CylinderCommand.EXTEND);
IF ext THEN
    _M_TagCommand(Id := 1, Label := 'std.command.clamp');
ELSE
    _M_TagCommand(Id := 2, Label := 'std.command.unclamp');
END_IF
CASE _step OF
    10:  // command both cylinders in parallel (Annex B)
        OutCmd.Confirmed := FALSE;
        CylA.Abort := FALSE;
        CylB.Abort := FALSE;
        CylA.Command := dir;
        CylB.Command := dir;
        CylA.Execute := TRUE;
        CylB.Execute := TRUE;
        _tSettle(IN := FALSE);
        _step := 20;
    20:  // join on both Done — roll up the first child Error, or its HELD reason (§8.2)
        IF CylA.Error OR CylB.Error THEN
            _M_RollupFault();
            CylA.Abort := TRUE;                    // stop the partner safely
            CylB.Abort := TRUE;
            CylA.Execute := FALSE;
            CylB.Execute := FALSE;
        ELSIF CylA.Held OR CylB.Held THEN
            // §6.1 HELD — a child is waiting on a named condition, not broken. Keep
            // the join open and adopt its reason so the EM is held-and-explained
            // instead of silently BUSY; both children resume by themselves. The
            // partner keeps its command: aborting it would turn a recoverable wait
            // into the half-finished clamp this join exists to prevent.
            _M_RollupHold();
        ELSIF CylA.Done AND CylB.Done THEN
            CylA.Execute := FALSE;
            CylB.Execute := FALSE;
            _step := 30;
        END_IF
    30:  // settle, then confirm both feedbacks held (EM-level check, Annex B)
        _tSettle(IN := TRUE, PT := ParCfg.SettleTime);
        IF _tSettle.Q THEN
            _tSettle(IN := FALSE);
            IF (ext AND CylA.OutImm.Extended AND CylB.OutImm.Extended)
            OR ((NOT ext) AND CylA.OutImm.Retracted AND CylB.OutImm.Retracted) THEN
                OutImm.Clamped   := ext;
                OutImm.Unclamped := NOT ext;
                OutCmd.Confirmed := TRUE;
                _M_Complete();
            ELSE
                _M_FaultN(PL_ModuleReasons.CLAMP_NOT_CONFIRMED, 'std.error.clampNotConfirmedAfterSettle');
            END_IF
        END_IF
ELSE
    _M_Fault(E_Reason.STEP_STALLED, 'std.error.undefinedStep');
END_CASE
END_METHOD

END_FUNCTION_BLOCK

// ---- FB_CylinderCM.TcPOU
// Annex A/B pattern on the base class: the type is ONLY its device logic.
FUNCTION_BLOCK FB_CylinderCM EXTENDS FB_ControlModuleBase
VAR_INPUT
    Command : E_CylinderCommand;
    ParCfg : ST_CylinderParCfg;
    ParCmd : ST_CylinderParCmd;
END_VAR
VAR_OUTPUT
    OutCmd : ST_CylinderOutCmd;
    OutImm : ST_CylinderOutImm;
    Intlk  : FB_PermIntlk;
END_VAR
VAR
    {attribute 'OPC.UA.DA' := '0'}
    _hal    : REFERENCE TO ST_CylinderHal;
    {attribute 'OPC.UA.DA' := '0'}
    _recipe : I_RecipeProvider;
    _tMove  : TON;
    _areaSafe : BOOL := TRUE;           // §7.2 application-supplied area/process interlock
    _areaSafeKey : STRING(255);
    _parCfgStaged : ST_CylinderParCfg;
    _recipePrepared : BOOL;
    _directionPermitsConfigured : BOOL;
    _extendPermit, _retractPermit : BOOL := TRUE;
    _extendPermitKey, _retractPermitKey : STRING(255);
    _extendedSensorTag, _retractedSensorTag : STRING(80);
    _extendedSensorAddress, _retractedSensorAddress : STRING(80);
    _extendOutputTag, _retractOutputTag : STRING(80);
    _extendedTimeoutKey, _retractedTimeoutKey, _bothSensorsKey : STRING(255);
    _bothSensorTags, _bothSensorAddresses : STRING(80);
END_VAR

Cyclic();

METHOD PROTECTED OnCyclic : DINT
OnCyclic := SUPER^.OnCyclic();
Intlk.Cond[1] := _areaSafe;             // §7.2 area-safe/air-ok, supplied via SetAreaSafe
IF NOT _directionPermitsConfigured OR (Command = E_CylinderCommand.NONE) THEN
    Intlk.Cond[2] := TRUE;
ELSIF Command = E_CylinderCommand.EXTEND THEN
    Intlk.Cond[2] := _extendPermit;
ELSIF Command = E_CylinderCommand.RETRACT THEN
    Intlk.Cond[2] := _retractPermit;
ELSE
    Intlk.Cond[2] := FALSE;
END_IF
Intlk();
IF __ISVALIDREF(_hal) THEN              // defensive (§5.6) [TC3]
    OutImm.Extended  := _hal.ExtendedFb;
    OutImm.Retracted := _hal.RetractedFb;
END_IF
OutImm.ExtendedSensorTag := _extendedSensorTag;
OutImm.RetractedSensorTag := _retractedSensorTag;
OutImm.ExtendOutputTag := _extendOutputTag;
OutImm.RetractOutputTag := _retractOutputTag;
END_METHOD

// Schematic identity is application configuration, not device behavior.
// Diagnostics keep SourcePath as this module and add the exact failed channel.
METHOD ConfigureIoIdentity
VAR_INPUT
    Identity : ST_CylinderIoIdentity;
END_VAR
_extendedSensorTag := Identity.ExtendedSensor.Tag;
_extendedSensorAddress := Identity.ExtendedSensor.Address;
_retractedSensorTag := Identity.RetractedSensor.Tag;
_retractedSensorAddress := Identity.RetractedSensor.Address;
_extendOutputTag := Identity.ExtendOutput.Tag;
_retractOutputTag := Identity.RetractOutput.Tag;
_extendedTimeoutKey := Identity.ExtendedTimeoutKey;
_retractedTimeoutKey := Identity.RetractedTimeoutKey;
_bothSensorsKey := Identity.BothSensorsKey;
_bothSensorTags := CONCAT(Identity.ExtendedSensor.Tag, CONCAT(' / ', Identity.RetractedSensor.Tag));
_bothSensorAddresses := CONCAT(Identity.ExtendedSensor.Address, CONCAT(' / ', Identity.RetractedSensor.Address));
END_METHOD

// Functional stop used by an owning sequence on abort/interlock loss.
// This is not a certified stop; the safety system remains authoritative.
METHOD WithdrawOutputs
IF __ISVALIDREF(_hal) THEN
    _hal.ExtendOut := FALSE;
    _hal.RetractOut := FALSE;
END_IF
END_METHOD

// Symmetric counterpart to WithdrawOutputs, for an owning sequence that withdrew a
// cylinder to hold a phase and now wants it driving again — a press dwell whose
// two-hand button was released and re-pressed, where the force comes from the valve
// latched by the already-completed EXTEND, so nothing else would re-energize it.
// Re-asserts ONLY the last commanded direction and ONLY while that direction's own
// permit is satisfied, so it can never restore an output the interlock is withholding:
// the caller asks, this module still decides. Idempotent; safe to call every scan.
// Not a certified enable — the safety system remains authoritative (§9).
METHOD RestoreOutputs
VAR
    permitted : BOOL;
END_VAR
IF NOT __ISVALIDREF(_hal) THEN
    RETURN;
END_IF
IF Command = E_CylinderCommand.EXTEND THEN
    permitted := _extendPermit OR NOT _directionPermitsConfigured;
ELSIF Command = E_CylinderCommand.RETRACT THEN
    permitted := _retractPermit OR NOT _directionPermitsConfigured;
ELSE
    permitted := FALSE;                 // no direction commanded: nothing to restore (§5.6)
END_IF
IF NOT permitted OR NOT Intlk.AllOk THEN
    RETURN;
END_IF
_hal.ExtendOut  := (Command = E_CylinderCommand.EXTEND);
_hal.RetractOut := (Command = E_CylinderCommand.RETRACT);
END_METHOD

METHOD PROTECTED OnAbort : DINT
OnAbort := SUPER^.OnAbort();            // base first (§3.14.2)
IF __ISVALIDREF(_hal) THEN
    _hal.ExtendOut := FALSE;
    _hal.RetractOut := FALSE;
END_IF
END_METHOD

METHOD PrepareRecipe : BOOL
VAR_INPUT
    Model : ST_ModelId;
END_VAR
IF _recipe = 0 THEN
    _parCfgStaged := ParCfg;
    _recipePrepared := TRUE;
    PrepareRecipe := TRUE;
ELSIF _recipe.Load(ModelCode := Model.ModelCode, RecipeKey := 'CylinderCM', pParCfg := ADR(_parCfgStaged), Size := SIZEOF(_parCfgStaged)) THEN
    _recipePrepared := TRUE;
    PrepareRecipe := TRUE;
ELSE
    _M_Fault(E_Reason.RECIPE_INVALID, 'std.error.recipeSchemaInvalid');
    _recipePrepared := FALSE;
    PrepareRecipe := FALSE;
END_IF
END_METHOD

METHOD CommitRecipe
IF _recipePrepared THEN ParCfg := _parCfgStaged; END_IF
_recipePrepared := FALSE;
END_METHOD

METHOD AbortRecipe
_recipePrepared := FALSE;
END_METHOD

METHOD Setup : BOOL
VAR_INPUT
    Name   : STRING(80);
    HalRef : REFERENCE TO ST_CylinderHal;
    Recipe : I_RecipeProvider;
END_VAR
VAR
    InitialModel : ST_ModelId;
END_VAR
_M_SetName(Name);
_M_SetPresentation(DisplayNameKey := 'std.moduleType.cylinder.name', DescriptionKey := 'std.moduleType.cylinder.description', TypeKey := 'std.moduleType.cylinder');
_hal REF= HalRef;                        // [TC3] TC3 §3.11
_recipe := Recipe;
// A library type owns a std.* key; an application overrides the text through
// SetAreaSafe when its own condition is more specific (§7.2.1).
Intlk.Define(Index := 1, Description := 'std.interlock.areaSafe', Reason := E_Reason.INTERLOCK_DROPPED, Bypassable := FALSE);
Intlk.Define(Index := 2, Description := 'std.interlock.directionPermitted', Reason := E_Reason.INTERLOCK_DROPPED, Bypassable := FALSE);
_M_PublishCommand(Value := TO_DINT(E_CylinderCommand.EXTEND), Label := 'std.command.extend');
_M_PublishCommand(Value := TO_DINT(E_CylinderCommand.RETRACT), Label := 'std.command.retract');
Setup := PrepareRecipe(Model := InitialModel);
IF Setup THEN CommitRecipe(); END_IF
END_METHOD

// Core §7.2/§7.2.1 — the application supplies this type's area/process interlock,
// the same shape as SetDirectionalPermits: a method (not an OPC UA write), and the
// condition is re-evaluated every scan so a manual command obeys the same rule.
//
// This replaces a SIM-only force hook that used to drive Cond[1] directly. That
// hook was the ONLY writer of the condition, so the slot an operator sees as
// "area safe" could be moved by a test and by nothing else: a reusable type
// published an interlock its application had no way to supply (§7.2.1), and the
// bypass shipped in every release build (§5.7). Driving the real condition is
// also strictly better test evidence - T3 now exercises the shipped path.
//
// Defaults TRUE: a station that declares no area interlock is not gated by one.
METHOD SetAreaSafe
VAR_INPUT
    Ok : BOOL;
    DescriptionKey : STRING(255);
END_VAR
_areaSafe := Ok;
_areaSafeKey := DescriptionKey;
IF _areaSafeKey <> '' THEN
    Intlk.Define(Index := 1, Description := _areaSafeKey, Reason := E_Reason.INTERLOCK_DROPPED, Bypassable := FALSE);
ELSE
    ;
END_IF
END_METHOD

METHOD PROTECTED _M_Dispatch
VAR
    ext : BOOL;
    d   : ST_Diagnostic;
END_VAR
IF _manualReq THEN
    _manualReq := FALSE;
    IF (_manualCmd = TO_DINT(E_CylinderCommand.EXTEND)) OR (_manualCmd = TO_DINT(E_CylinderCommand.RETRACT)) THEN
        Command := _manualCmd;
    ELSE
        _M_Fault(E_Reason.UNSUPPORTED_COMMAND, 'std.error.unsupportedCylinderCommand');
        RETURN;
    END_IF
END_IF
IF (Command <> E_CylinderCommand.EXTEND) AND (Command <> E_CylinderCommand.RETRACT) THEN
    _M_Fault(E_Reason.UNSUPPORTED_COMMAND, 'std.error.unsupportedCylinderCommand');
    RETURN;
END_IF
IF Command = E_CylinderCommand.EXTEND THEN
    _M_TagCommand(Id := 1, Label := 'std.command.extend');       // §8.11.4(a)
    IF _directionPermitsConfigured THEN
        Intlk.Define(Index := 2, Description := _extendPermitKey, Reason := E_Reason.INTERLOCK_DROPPED, Bypassable := FALSE);
        Intlk.Cond[2] := _extendPermit;
    ELSE
        Intlk.Cond[2] := TRUE;
    END_IF
ELSE
    _M_TagCommand(Id := 2, Label := 'std.command.retract');
    IF _directionPermitsConfigured THEN
        Intlk.Define(Index := 2, Description := _retractPermitKey, Reason := E_Reason.INTERLOCK_DROPPED, Bypassable := FALSE);
        Intlk.Cond[2] := _retractPermit;
    ELSE
        Intlk.Cond[2] := TRUE;
    END_IF
END_IF
Intlk();
IF NOT Intlk.AllOk THEN
    // §6.1 HELD, not a fault. An interlock is by definition a condition that must
    // hold DURING motion, and losing one is often expected operator behaviour —
    // releasing a two-hand button is the designed way to stop a stroke. Faulting
    // classified that as a defect and forced the ABORTED/STOPPED exit (Reset ->
    // IDLE), which on the press was unreachable: the fault's own condition included
    // "two-hand held during a stroke", which can only be restored by running.
    // Nothing is weakened here — the output is withdrawn in the same place, by the
    // same permit — only the classification and the way out change: the module stays
    // BUSY with its outputs off and resumes when the condition returns (§8.4: this
    // is a wait, not a downtime event). Rewinding to N010 means the resume
    // re-energizes the direction output and re-arms MoveTimeout with a full window,
    // so a hold cannot silently consume the travel time it was not moving for.
    _hal.ExtendOut := FALSE;
    _hal.RetractOut := FALSE;
    d := Intlk.Diagnostic;
    d.SourcePath := _name;                            // owner sets the path (§7.2)
    _M_HoldDiag(Diag := d);
    _step := 10;
    RETURN;
END_IF
IF _hal.ExtendedFb AND _hal.RetractedFb THEN
    IF _bothSensorsKey <> '' THEN
        _M_FaultIoN(Code := PL_ModuleReasons.CYL_BOTH_SENSORS, Text := _bothSensorsKey,
            IoTag := _bothSensorTags, IoAddress := _bothSensorAddresses);
    ELSE
        _M_FaultN(Code := PL_ModuleReasons.CYL_BOTH_SENSORS, Text := 'std.error.cylinderBothSensors');
    END_IF
    RETURN;
END_IF
ext := (Command = E_CylinderCommand.EXTEND);
CASE _step OF
    10:
        OutCmd.Reached := FALSE;
        _hal.ExtendOut  := ext;
        _hal.RetractOut := NOT ext;
        _tMove(IN := FALSE);
        _step := 20;
    20:
        _tMove(IN := TRUE, PT := ParCfg.MoveTimeout);
        IF (ext AND _hal.ExtendedFb) OR ((NOT ext) AND _hal.RetractedFb) THEN
            _tMove(IN := FALSE);
            OutCmd.Reached := TRUE;
            _M_Complete();
        ELSIF _tMove.Q THEN
            _tMove(IN := FALSE);
            IF ext AND (_extendedSensorTag <> '') THEN
                _M_FaultIoN(Code := PL_ModuleReasons.CYL_NOT_EXTENDED, Text := _extendedTimeoutKey,
                    IoTag := _extendedSensorTag, IoAddress := _extendedSensorAddress);
            ELSIF (NOT ext) AND (_retractedSensorTag <> '') THEN
                _M_FaultIoN(Code := PL_ModuleReasons.CYL_NOT_RETRACTED, Text := _retractedTimeoutKey,
                    IoTag := _retractedSensorTag, IoAddress := _retractedSensorAddress);
            ELSIF ext THEN
                _M_FaultN(Code := PL_ModuleReasons.CYL_NOT_EXTENDED, Text := 'std.error.cylinderExtendTimeout');
            ELSE
                _M_FaultN(Code := PL_ModuleReasons.CYL_NOT_RETRACTED, Text := 'std.error.cylinderRetractTimeout');
            END_IF
        END_IF
ELSE
    _M_Fault(E_Reason.STEP_STALLED, 'std.error.undefinedStep');    // defined ELSE (§5.6)
END_CASE
END_METHOD

// Functional collision/process interlocks supplied by the owning EM/Unit.
// Methods are not OPC UA writes; the check is repeated inside dispatch so manual
// commands use the same rule. Certified safety remains external.
METHOD SetDirectionalPermits
VAR_INPUT
    ExtendOk : BOOL;
    RetractOk : BOOL;
    ExtendDescriptionKey : STRING(255);
    RetractDescriptionKey : STRING(255);
END_VAR
_directionPermitsConfigured := TRUE;
_extendPermit := ExtendOk;
_retractPermit := RetractOk;
_extendPermitKey := ExtendDescriptionKey;
_retractPermitKey := RetractDescriptionKey;
END_METHOD

// Pure release-query companion to SetDirectionalPermits. The owning Unit uses
// this for act-or-explain so the HMI checks the exact permit used by dispatch.
METHOD AppendDirectionalRelease : INT
VAR_INPUT
    Value : DINT;
END_VAR
VAR_IN_OUT
    Report : ST_ReleaseReport;
END_VAR
VAR
    permitted : BOOL;
    validCommand : BOOL;
    descriptionKey : STRING(255);
END_VAR
permitted := TRUE;
validCommand := (Value = TO_DINT(E_CylinderCommand.EXTEND))
    OR (Value = TO_DINT(E_CylinderCommand.RETRACT));
descriptionKey := '';
IF _directionPermitsConfigured AND (Value = TO_DINT(E_CylinderCommand.EXTEND)) THEN
    permitted := _extendPermit;
    descriptionKey := _extendPermitKey;
ELSIF _directionPermitsConfigured AND (Value = TO_DINT(E_CylinderCommand.RETRACT)) THEN
    permitted := _retractPermit;
    descriptionKey := _retractPermitKey;
ELSIF NOT validCommand THEN
    permitted := FALSE;
    descriptionKey := 'std.error.unsupportedCylinderCommand';
ELSE
    permitted := TRUE;
END_IF
IF NOT permitted AND (Report.Count < PL_Fraktal.MAX_RELEASE_REASONS) THEN
    Report.Count := Report.Count + 1;
    Report.Reasons[Report.Count].Description := descriptionKey;
    Report.Reasons[Report.Count].SourcePath := _name;
    IF validCommand THEN
        Report.Reasons[Report.Count].ReasonCode := E_Reason.INTERLOCK_DROPPED;
    ELSE
        Report.Reasons[Report.Count].ReasonCode := E_Reason.UNSUPPORTED_COMMAND;
    END_IF
    Report.Reasons[Report.Count].Kind := E_ReleaseKind.INTERLOCK;
    Report.Reasons[Report.Count].Bypassable := FALSE;
END_IF
AppendDirectionalRelease := Report.Count;
END_METHOD

END_FUNCTION_BLOCK

// ---- FB_DigitalInputCM.TcPOU
// Basic passive digital-input CM. Owning logic consumes semantic Value; the
// project catalog injects the physical identity separately from the HAL.
FUNCTION_BLOCK FB_DigitalInputCM EXTENDS FB_ControlModuleBase
VAR_INPUT
    ParCfg : ST_DigitalInputParCfg;
    ParCmd : ST_DigitalInputParCmd;
END_VAR
VAR_OUTPUT
    OutCmd : ST_DigitalInputOutCmd;
    OutImm : ST_DigitalInputOutImm;
END_VAR
VAR
    {attribute 'OPC.UA.DA' := '0'}
    _hal : REFERENCE TO ST_DigitalInputHal;
    _identity : ST_IoPointIdentity;
END_VAR

Cyclic();

METHOD Setup : BOOL
VAR_INPUT
    Name : STRING(80);
    HalRef : REFERENCE TO ST_DigitalInputHal;
    DisplayNameKey : STRING(160);
    DescriptionKey : STRING(160);
END_VAR
_M_SetName(Name);
_M_SetPresentation(DisplayNameKey := DisplayNameKey, DescriptionKey := DescriptionKey, TypeKey := 'std.moduleType.digitalInput');
_hal REF= HalRef;
Setup := __ISVALIDREF(_hal);
END_METHOD

METHOD ConfigureIoIdentity
VAR_INPUT
    Identity : ST_IoPointIdentity;
END_VAR
_identity := Identity;
END_METHOD

METHOD PROTECTED OnCyclic : DINT
OnCyclic := SUPER^.OnCyclic();
IF __ISVALIDREF(_hal) THEN
    OutImm.Value := _hal.Value;
    OutImm.Quality := _hal.Quality;
ELSE
    OutImm.Value := FALSE;
    OutImm.Quality := FALSE;
END_IF
OutImm.IoTag := _identity.Tag;
END_METHOD

METHOD PROTECTED _M_Dispatch
_M_Fault(E_Reason.UNSUPPORTED_COMMAND,
    'std.error.passiveInputHasNoCommand');
END_METHOD

END_FUNCTION_BLOCK

// ---- FB_AirPressureMonitorCM.TcPOU
// Basic passive two-threshold pneumatic-pressure CM. Both switches active is
// implausible and faults with both exact tags; neither/high-only are status states.
FUNCTION_BLOCK FB_AirPressureMonitorCM EXTENDS FB_ControlModuleBase
VAR_INPUT
    ParCfg : ST_AirPressureParCfg;
    ParCmd : ST_AirPressureParCmd;
END_VAR
VAR_OUTPUT
    OutCmd : ST_AirPressureOutCmd;
    OutImm : ST_AirPressureOutImm;
END_VAR
VAR
    {attribute 'OPC.UA.DA' := '0'}
    _hal : REFERENCE TO ST_AirPressureHal;
    _lowIdentity, _operatingIdentity : ST_IoPointIdentity;
    _bothTags, _bothAddresses : STRING(80);
    // Both switches reading active is only a genuine wiring/sensor fault when it
    // PERSISTS. The two mechanical switches trip at different pressures and have
    // their own response delays, so while the system pressurises a brief overlap
    // is normal physics, not a defect. Because the fault latches (an operator
    // reset is required to clear it), a single spurious cycle would otherwise
    // block Control On indefinitely — observed on the press, where the sensors
    // read consistently in steady state yet the conflict fault stayed raised.
    // Same idiom as ST_ConfigurableCylinderParCfg.DiscrepancyTime.
    _conflictTimer : TON;
END_VAR
VAR PERSISTENT
    // §3.8a/§3.8b — deployment data: editable from the HMI, retained across
    // a restart, and never part of a model recipe. The Setup registration,
    // not this declaration, is what permits a write (§3.10.2).
    StationCfg : ST_AirPressureStationCfg;
END_VAR

Cyclic();

METHOD Setup : BOOL
VAR_INPUT
    Name : STRING(80);
    HalRef : REFERENCE TO ST_AirPressureHal;
END_VAR
_M_SetName(Name);
_M_SetPresentation(DisplayNameKey := 'std.moduleType.airPressure.name',
    DescriptionKey := 'std.moduleType.airPressure.description',
    TypeKey := 'std.moduleType.airPressure');
_hal REF= HalRef;
// §3.8b — a retained image from an unrecognized layout is re-initialized,
// never interpreted by field position. Version 0 is a first boot: nothing
// was retained, so nothing was lost and nothing is announced.
IF StationCfg.SchemaVersion <> 1 THEN
    StationCfg.SchemaVersion := 1;
    StationCfg.ConflictTime := T#500MS;
END_IF
// §3.10.2 — publish the one value a commissioning engineer tunes here.
// READY is required: re-timing fault qualification underneath a running
// cycle would change what counts as a fault while it is being judged.
Setup := __ISVALIDREF(_hal)
    AND M_RegisterConfigDuration(Key := 'airPressure.conflictTime',
        Item := 'StationCfg/ConflictTime',
        LabelKey := 'std.config.airPressure.conflictTime',
        Kind := E_ConfigKind.STATION_CFG,
        pTarget := ADR(StationCfg.ConflictTime),
        MinimumMs := 0, MaximumMs := 10000,
        RequiresReady := TRUE);
END_METHOD

METHOD ConfigureIoIdentity
VAR_INPUT
    LowSensor : ST_IoPointIdentity;
    OperatingSensor : ST_IoPointIdentity;
END_VAR
_lowIdentity := LowSensor;
_operatingIdentity := OperatingSensor;
_bothTags := CONCAT(LowSensor.Tag, CONCAT(' / ', OperatingSensor.Tag));
_bothAddresses := CONCAT(LowSensor.Address, CONCAT(' / ', OperatingSensor.Address));
END_METHOD

METHOD PROTECTED OnCyclic : DINT
OnCyclic := SUPER^.OnCyclic();
IF __ISVALIDREF(_hal) THEN
    OutImm.LowPressure := _hal.LowPressure;
    OutImm.OperatingPressure := _hal.OperatingPressure;
    OutImm.Quality := _hal.Quality;
    // Qualify the conflict over StationCfg.ConflictTime before treating it as
    // a fault, so the transient overlap seen while air fills cannot latch a
    // permanent fault.
    _conflictTimer(IN := _hal.LowPressure AND _hal.OperatingPressure,
        PT := StationCfg.ConflictTime);
    OutImm.Contradictory := _conflictTimer.Q;
    OutImm.PressureOk := _hal.OperatingPressure AND NOT _hal.LowPressure AND _hal.Quality;
    IF OutImm.Contradictory THEN
        _M_FaultIoN(Code := PL_ModuleReasons.AIR_SWITCH_CONFLICT,
            Text := 'std.error.airPressureSwitchConflict',
            IoTag := _bothTags, IoAddress := _bothAddresses);
    END_IF
ELSE
    OutImm.LowPressure := FALSE;
    OutImm.OperatingPressure := FALSE;
    OutImm.Quality := FALSE;
    OutImm.Contradictory := FALSE;
    OutImm.PressureOk := FALSE;
END_IF
OutImm.LowSensorTag := _lowIdentity.Tag;
OutImm.OperatingSensorTag := _operatingIdentity.Tag;
END_METHOD

METHOD PROTECTED _M_Dispatch
_M_Fault(E_Reason.UNSUPPORTED_COMMAND,
    'std.error.passiveInputHasNoCommand');
END_METHOD

END_FUNCTION_BLOCK

// ---- FB_CylinderSim.TcPOU
// §5.7 per-type sim plant model: drives the HAL feedback with a travel time —
// shared by TcUnit suites and virtual commissioning (§2.6).
FUNCTION_BLOCK FB_CylinderSim
VAR
    Travel : TIME := T#0S;
END_VAR
VAR
    {attribute 'OPC.UA.DA' := '0'}
    _hal : REFERENCE TO ST_CylinderHal;
    _tE, _tR : TON;
END_VAR

IF NOT __ISVALIDREF(_hal) THEN
    RETURN;
END_IF
_tE(IN := _hal.ExtendOut AND NOT _hal.ExtendedFb, PT := Travel);
IF _tE.Q THEN
    _hal.ExtendedFb  := TRUE;
    _hal.RetractedFb := FALSE;
END_IF
_tR(IN := _hal.RetractOut AND NOT _hal.RetractedFb, PT := Travel);
IF _tR.Q THEN
    _hal.RetractedFb := TRUE;
    _hal.ExtendedFb  := FALSE;
END_IF

METHOD Setup : BOOL
VAR_INPUT
    HalRef : REFERENCE TO ST_CylinderHal;
    TravelTime : TIME;
END_VAR
_hal REF= HalRef;
Travel := TravelTime;
Setup := TRUE;
END_METHOD

END_FUNCTION_BLOCK

// ---- FB_PowerGroupCM.TcPOU
// §9.8 basic power-group CM. It requests functional enable; certified safety
// logic and field-output watchdogs remain authoritative. Recovery never self-energizes.
FUNCTION_BLOCK FB_PowerGroupCM EXTENDS FB_ControlModuleBase
VAR_INPUT
    Command : E_PowerGroupCommand;
    ParCfg  : ST_PowerGroupParCfg;
    ParCmd  : ST_PowerGroupParCmd;
END_VAR
VAR_OUTPUT
    OutCmd : ST_PowerGroupOutCmd;
    OutImm : ST_PowerGroupOutImm;
END_VAR
VAR
    {attribute 'OPC.UA.DA' := '0'}
    _hal : REFERENCE TO ST_PowerGroupHal;
    _tFeedback : TON;
    _rearmRequired : BOOL;
END_VAR

Cyclic();

METHOD Setup : BOOL
VAR_INPUT
    Name : STRING(80);
    HalRef : REFERENCE TO ST_PowerGroupHal;
END_VAR
_M_SetName(Name);
_M_SetPresentation(DisplayNameKey := 'std.moduleType.powerGroup.name', DescriptionKey := 'std.moduleType.powerGroup.description', TypeKey := 'std.moduleType.powerGroup');
_hal REF= HalRef;
// Power control deliberately has no MANUAL command catalog: it uses the Unit's
// POWER_CONTROL-gated ReqControlOn/ReqControlOff endpoint (§9.8).
Setup := TRUE;
END_METHOD

METHOD PROTECTED OnCyclic : DINT
VAR
    busMustDrop : BOOL;
END_VAR
OnCyclic := SUPER^.OnCyclic();
CASE ParCfg.FieldbusLossReaction OF
    E_FieldbusLossReaction.ALARM_ONLY, E_FieldbusLossReaction.STOP_UNIT:
        busMustDrop := FALSE;
    E_FieldbusLossReaction.POWER_GROUP_OFF, E_FieldbusLossReaction.CONTROL_OFF:
        busMustDrop := TRUE;
ELSE
    busMustDrop := TRUE; // unknown policy fails toward power removal
END_CASE
IF (NOT _hal.SafetyPermit) OR (busMustDrop AND NOT _hal.FieldbusHealthy) THEN
    IF _hal.EnableRequestOut OR _hal.PowerFeedback THEN _rearmRequired := TRUE; END_IF
    _hal.EnableRequestOut := FALSE;
END_IF
OutCmd.PowerOn := _hal.PowerFeedback;
OutImm.Status.Present := TRUE;
OutImm.Status.Name := _name;
OutImm.Status.Kind := ParCfg.Kind;
OutImm.Status.RequiredForControl := ParCfg.RequiredForControl;
OutImm.Status.RequestedOn := _hal.EnableRequestOut;
OutImm.Status.PowerOn := _hal.PowerFeedback;
OutImm.Status.SafetyPermit := _hal.SafetyPermit;
OutImm.Status.FieldbusHealthy := _hal.FieldbusHealthy;
OutImm.Status.FieldbusLossReaction := ParCfg.FieldbusLossReaction;
OutImm.Status.RearmRequired := _rearmRequired;
IF _hal.PowerFeedback THEN
    OutImm.Status.State := E_PowerState.ON;
ELSIF _rearmRequired THEN
    OutImm.Status.State := E_PowerState.TRIPPED;
ELSE
    OutImm.Status.State := E_PowerState.OFF;
END_IF
OutImm.Status.Diagnostic := Status.Diagnostic;
ControlPower.Present := TRUE;
ControlPower.GroupCount := 1;
ControlPower.Groups[1] := OutImm.Status;
ControlPower.RequestedOn := _hal.EnableRequestOut;
ControlPower.ControlOn := _hal.PowerFeedback;
ControlPower.RearmRequired := _rearmRequired;
END_METHOD

METHOD PROTECTED _M_Dispatch
IF _manualReq THEN
    Command := _manualCmd;
    _manualReq := FALSE;
END_IF
CASE _step OF
    10:
        CASE Command OF
            E_PowerGroupCommand.POWER_ON:
                IF (NOT _hal.SafetyPermit) OR (NOT _hal.FieldbusHealthy) THEN
                    _M_FaultN(Code := PL_ModuleReasons.POWER_ENABLE_WITHHELD, Text := 'std.error.powerEnableWithheld');
                ELSE
                    _rearmRequired := FALSE;
                    _hal.EnableRequestOut := TRUE;
                    _step := 20;
                END_IF
            E_PowerGroupCommand.POWER_OFF:
                _hal.EnableRequestOut := FALSE;
                _step := 30;
        ELSE
            _M_Fault(E_Reason.UNSUPPORTED_COMMAND, 'std.error.unsupportedPowerCommand');
        END_CASE
    20:
        _tFeedback(IN := NOT _hal.PowerFeedback, PT := ParCfg.FeedbackTimeout);
        IF _hal.PowerFeedback THEN _tFeedback(IN := FALSE); _M_Complete();
        ELSIF _tFeedback.Q THEN _M_FaultN(Code := PL_ModuleReasons.POWER_FEEDBACK_TIMEOUT, Text := 'std.error.powerOnFeedbackTimeout'); END_IF
    30:
        _tFeedback(IN := _hal.PowerFeedback, PT := ParCfg.FeedbackTimeout);
        IF NOT _hal.PowerFeedback THEN _tFeedback(IN := FALSE); _M_Complete();
        ELSIF _tFeedback.Q THEN _M_FaultN(Code := PL_ModuleReasons.POWER_FEEDBACK_TIMEOUT, Text := 'std.error.powerOffFeedbackTimeout'); END_IF
ELSE
    _hal.EnableRequestOut := FALSE;
    _M_Fault(E_Reason.STEP_STALLED, 'std.error.undefinedPowerStep');
END_CASE
END_METHOD

METHOD PROTECTED OnAbort : DINT
OnAbort := SUPER^.OnAbort();
_hal.EnableRequestOut := FALSE;
_rearmRequired := TRUE;
END_METHOD

END_FUNCTION_BLOCK

// ---- FB_TwoHandStartCM.TcPOU
// Functional cycle-start edge from a certified two-hand-control result.
// This CM does not implement simultaneity, anti-tie-down, PL or safe outputs.
FUNCTION_BLOCK FB_TwoHandStartCM EXTENDS FB_ControlModuleBase
VAR_INPUT
    ParCfg : ST_TwoHandParCfg;
    ParCmd : ST_TwoHandParCmd;
END_VAR
VAR_OUTPUT
    OutCmd : ST_TwoHandOutCmd;
    OutImm : ST_TwoHandOutImm;
END_VAR
VAR
    {attribute 'OPC.UA.DA' := '0'}
    _hal : REFERENCE TO ST_TwoHandHal;
    _safeRise : R_TRIG;
    _armed : BOOL;
END_VAR

Cyclic();

METHOD Setup : BOOL
VAR_INPUT
    Name : STRING(80);
    HalRef : REFERENCE TO ST_TwoHandHal;
END_VAR
_M_SetName(Name);
_M_SetPresentation(DisplayNameKey := 'std.moduleType.twoHand.name', DescriptionKey := 'std.moduleType.twoHand.description', TypeKey := 'std.moduleType.twoHand');
_hal REF= HalRef;
Setup := TRUE;
END_METHOD

METHOD PROTECTED OnCyclic : DINT
OnCyclic := SUPER^.OnCyclic();
OutImm.StartPulse := FALSE;
OutCmd.StartAccepted := FALSE;
IF __ISVALIDREF(_hal) THEN
    OutImm.LeftPressed := _hal.LeftPressed;
    OutImm.RightPressed := _hal.RightPressed;
    OutImm.FieldbusHealthy := _hal.FieldbusHealthy;
    OutImm.SafeActive := _hal.SafeActive AND _hal.FieldbusHealthy;
    IF NOT _hal.FieldbusHealthy THEN
        _armed := FALSE;
    ELSIF NOT _hal.LeftPressed AND NOT _hal.RightPressed AND NOT _hal.SafeActive THEN
        _armed := TRUE;
    END_IF
    _safeRise(CLK := OutImm.SafeActive);
    IF _safeRise.Q AND (_armed OR NOT ParCfg.RequireReleaseBetweenCycles) THEN
        OutImm.StartPulse := TRUE;
        OutCmd.StartAccepted := TRUE;
        _armed := FALSE;
    END_IF
ELSE
    OutImm.LeftPressed := FALSE;
    OutImm.RightPressed := FALSE;
    OutImm.SafeActive := FALSE;
    OutImm.FieldbusHealthy := FALSE;
    _armed := FALSE;
    _safeRise(CLK := FALSE);
END_IF
OutImm.Armed := _armed;
Safety.Present := TRUE;
Safety.AllSafe := OutImm.FieldbusHealthy;
Safety.DemandActive := OutImm.LeftPressed OR OutImm.RightPressed;
Safety.FaultActive := NOT OutImm.FieldbusHealthy;
Safety.DeviceCount := 1;
Safety.Devices[1].Present := TRUE;
Safety.Devices[1].Name := _name;
Safety.Devices[1].Kind := E_SafetyDeviceKind.TWO_HAND_CONTROL;
Safety.Devices[1].Ready := OutImm.Armed;
Safety.Devices[1].DemandActive := OutImm.LeftPressed OR OutImm.RightPressed;
Safety.Devices[1].SafeStateActive := NOT OutImm.SafeActive;
Safety.Devices[1].FieldbusHealthy := OutImm.FieldbusHealthy;
Safety.Devices[1].Description := 'std.safety.twoHandControl';
END_METHOD

METHOD PROTECTED _M_Dispatch
_M_Fault(E_Reason.UNSUPPORTED_COMMAND, 'std.error.twoHandHasNoCommand');
END_METHOD

END_FUNCTION_BLOCK
